FUNCTION_BLOCK Write_Register (* Template for a Simple Function Block Type *)
  (* Standard: 61499-1 *)
  (* Version 1.0, 2024-07-26, david *)
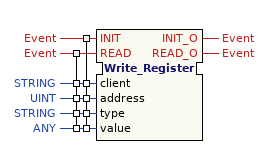
  EVENT_INPUT
    INIT WITH client, address, type, value; (* Initialization event *)
    READ WITH type, address, client, value; (* Read event *)
  END_EVENT
  EVENT_OUTPUT
    INIT_O; (* Init event out *)
    READ_O; (* Read event out *)
  END_EVENT
  VAR_INPUT
    client : STRING; (* client object *)
    address : UINT; (* register address *)
    type : STRING := INT; (* Datatype of register *)
    value : ANY; (* Value to be written *)
  END_VAR
END_FUNCTION_BLOCK
